(* IEC 61131-3 sources: SRCI/RobotLibrary/Library/POUs/BasicMove/MC_GroupInterrupt, 1 file *)

(* ---- MC_GroupInterruptFB.st ---- *)
/// Interrupt active movement, possible to continue movement
FUNCTION_BLOCK MC_GroupInterruptFB EXTENDS RobotLibraryBaseExecuteFB
// -------------------------------------------------------------------------
//  SRCI Robot Library
// -------------------------------------------------------------------------
//
//  Object:      GroupInterruptFB
//  Author:      Thorsten Brach
//  Date:        2024-06-01
//
//  Description:
//
//
//  Copyright:
//    (C) 2024 Thorsten Brach. All rights reserved
//             Licensed under the LGPL-3.0 license.
//
//  Disclaimer:
//    This project is provided without any guarantee and can be used for
//    private and commercial purposes. Any use is at the user’s
//    own risk and responsibility.
//
// -------------------------------------------------------------------------
VAR_INPUT
  /// Command parameter
  ParCmd          : GroupInterruptParCmd;
END_VAR

VAR_OUTPUT
  /// Command is transferred and confirmed by the RC
  CommandBuffered : BOOL;
  /// The command takes control of the motion of the according axis group.
  Active          : BOOL;
  /// Command output
  OutCmd          : GroupInterruptOutCmd;
END_VAR

VAR
  /// internal copy of command parameter
 _parCmd          : GroupInterruptParCmd;
  /// command data to send
 _command         : GroupInterruptSendData;
  /// response data received
 _response        : GroupInterruptRecvData;
END_VAR

  SUPER^(AxesGroup := AxesGroup);

END_FUNCTION_BLOCK

METHOD INTERNAL CheckAddParameter : BOOL
VAR_INPUT
  /// Payload pointer
  PayloadPtr : UDINT;
END_VAR
VAR
  /// Payload as byte array
  Payload    : ARRAY [1..SIZEOF(_command)] OF BYTE;
  /// Null Byte array
  Null       : ARRAY [1..SIZEOF(_command)] OF BYTE;
  /// Data length to compare
  DataLen    : UDINT;
END_VAR

  // Payload pointer must be decreased by one byte, because ADR(Payload) is already one byte !
  PayloadPtr := LIMIT (0, PayloadPtr - 1, SIZEOF(Payload) -1);
  // Convert command struct to payload array
  SysDepMemCpy( pDest := ADR(Payload), pSrc := ADR(_command), DataLen := SIZEOF(_command));
  // Calculate the data length to compare - at least one byte must be compared !
  DataLen := LIMIT(1, SIZEOF(Payload) - PayloadPtr, SIZEOF(Payload));
  // Compare Payload-Array with Null-Byte-Array
  CheckAddParameter := SysDepMemCmp( pData1 := ADR(Payload) + PayloadPtr , pData2 := ADR(Null), DataLen := DataLen) <>  RobotLibraryConstants.OK ;

END_METHOD

METHOD PROTECTED CheckFunctionSupported : BOOL
VAR_IN_OUT
  /// Robot assignment of function
  AxesGroup : AxesGroup;
END_VAR

  CheckFunctionSupported := AxesGroup.State.RobotData.RCSupportedFunctions.GroupInterrupt;

  IF ( NOT CheckFunctionSupported )
  THEN
    // call base implementation for set error and create log entry
    SUPER^.CheckFunctionSupported(AxesGroup := AxesGroup);
  END_IF

END_METHOD

METHOD PROTECTED CheckParameterChanged : BOOL
VAR_IN_OUT
  /// Robot assignment of function
  AxesGroup    : AxesGroup;
END_VAR

  // Check ParCmd Size is > 0, because MemCmp does not work correctly with size = 0
  IF (SIZEOF(ParCmd) = 0) OR (_stepCmd = 0)
  THEN
    RETURN;
  END_IF

  // compare memory
  _parameterChanged := ( SysDepMemCmp(pData1 := ADR(ParCmd), pData2 := ADR(_parCmd), DataLen := SIZEOF(ParCmd)) <> RobotLibraryConstants.OK );

  // check parameter valid ?
  _parameterValid   := CheckParameterValid( AxesGroup := AxesGroup );

  IF ((  _parameterChanged        )  AND
      (  _parameterValid          )) OR
      (  _parameterUpdateInternal )
  THEN
    // reset internal flag for send parameter update
   _parameterUpdateInternal := FALSE;
    // update internal copy of parameters
   _parCmd := ParCmd;
    // inc parameter sequence
   _command.ParSeq := _command.ParSeq + 1;
    // update command data
    CommandData := CreateCommandPayload(AxesGroup := AxesGroup); // ( Access via reference to rCommandFB in ACR )
    // notify active command register
    AxesGroup.Acyclic.ActiveCommandRegister.NotifyParameterChanged := _uniqueID;
  END_IF

END_METHOD

METHOD INTERNAL CreateCommandPayload : RobotLibraryCommandDataFB
VAR_IN_OUT
  /// Robot assignment of function
  AxesGroup : AxesGroup;
END_VAR
VAR
  /// Parameter count
 _parameterCnt : DINT;
END_VAR
// Table 6-273: Sent CMD payload (PLC to RC) of "GroupInterrupt"
// --------------------------
// Header
// --------------------------
// Byte 00 : UINT  - Type HB
// Byte 01 :       - Type LB
// Byte 02 : USINT - Reserve | ExecutionMode
// Byte 03 : USINT - ParSeq  | Priority
// --------------------------

  // set command parameter
  _command.CmdTyp     :=  CmdType.GroupInterrupt;
  _command.ExecMode   :=  ExecMode;
  _command.ParSeq     := _command.ParSeq;
  _command.Priority   :=  Priority;

  // copy command data to header
  _cmdHeader := _command;
  // call base implementation to copy header to payload buffer
  CreateCommandPayload := SUPER^.CreateCommandPayload(AxesGroup := AxesGroup);

  // Create logging
  CreateCommandPayloadLog(AxesGroup := AxesGroup, ParameterCnt := _parameterCnt);

END_METHOD

METHOD INTERNAL CreateCommandPayloadLog
VAR_IN_OUT
  /// Robot assignment of function
  AxesGroup : AxesGroup;
END_VAR
VAR_INPUT
  /// Parameter count
  ParameterCnt : DINT;
END_VAR

  // Create log entry for Parameter start
  CreateLogMessagePara1 ( Timestamp   := AxesGroup.State.SystemTime,
                          MessageType := MessageType.CMD,
                          Severity    := Severity.DEBUG,
                          MessageCode := 0,
                          MessageText := 'Create command payload with the {1} parameter(s) :',
                          Para1       := DINT_TO_STRING(ParameterCnt));

END_METHOD

METHOD FB_init : BOOL
VAR_INPUT
  /// if TRUE, the retain variables are initialized (warm start / cold start)
  bInitRetains : BOOL;
  /// if TRUE, the instance afterwards gets moved into the copy code (online change)
  bInCopyCode  : BOOL;
END_VAR

  MyType := 'MC_GroupInterruptFB';

  ExecMode := ExecutionMode.PARALLEL;
  Priority := PriorityLevel.NORMAL;

END_METHOD

METHOD PROTECTED OnExecRun : DINT
VAR_IN_OUT
  /// Robot assignment of function
  AxesGroup : AxesGroup;
END_VAR

  // call base implementation
  SUPER^.OnExecRun(AxesGroup := AxesGroup);

  CASE _stepCmd OF

    00:  IF ( _execute_R.Q ) AND ( NOT Error)
         THEN
           // Check function is supported and parameter are valid ?
           IF (( CheckFunctionSupported( AxesGroup := AxesGroup )) AND
               ( CheckParameterValid   ( AxesGroup := AxesGroup )))
           THEN
             // inc fast stop counter
             AxesGroup.Cyclic.PlcToRob.FastStop := AxesGroup.Cyclic.PlcToRob.FastStop + 1;
             // set busy flag
             Busy := TRUE;
             // Reset command outputs
             SysDepMemSet(pDest := ADR(OutCmd), Value := 0, DataLen := SIZEOF(OutCmd));
             // apply command parameter
            _parCmd := ParCmd;
             // init parameter sequence
            _command.ParSeq := 1;
             // create command data
             CommandData := CreateCommandPayload(AxesGroup := AxesGroup);
             // Add command to active command register
            _uniqueID := AxesGroup.Acyclic.ActiveCommandRegister.AddCmd( pCommandFB := ADR(THIS^ ));
             // set timeout
             SetTimeout(PT := _timeoutCmd, rTimer := _timerCmd);
             // inc step counter
            _stepCmd := _stepCmd + 1;
           END_IF
         END_IF

    01:  // Wait for responce received
         IF ( _responseReceived )
         THEN
           // reset response received flag
          _responseReceived := FALSE;
           // reset Active flag
           Active := FALSE;

           CASE  _response.State
           OF
             CmdMessageState.BUFFERED    : CommandBuffered := TRUE;
             CmdMessageState.ACTIVE      : Active          := TRUE;
             CmdMessageState.ERROR       : Error           := TRUE;
             CmdMessageState.DONE        : Done            := TRUE;

           END_CASE

           // Done, Aborted or Error ?
           IF (_response.State >= CmdMessageState.DONE )
           THEN
             // reset busy flag
             Busy := FALSE;
             // set timeout
             SetTimeout(PT := _timeoutCmd, rTimer := _timerCmd);
             // inc step counter
            _stepCmd := _stepCmd + 1;
           END_IF
         END_IF

    02: IF ( NOT Execute)
        THEN
          Reset();
        END_IF
  ELSE
    // invalid step
    ErrorID := RobotLibraryErrorIdEnum.ERR_INVALID_STEP;
  END_CASE

  // Reset FB
  IF ( NOT Execute )
  THEN
    Reset();
  END_IF

END_METHOD

METHOD INTERNAL ParseResponsePayload : DINT
VAR_INPUT
  /// Response data
  ResponseData : RobotLibraryResponseDataFB;
  /// Timestamp
  Timestamp    : SystemTime;
END_VAR
VAR
  /// Parameter count
 _parameterCnt : DINT;
END_VAR
// Table 6-274: Received CMD payload (RC to PLC) of "GroupInterrupt"
// --------------------------
// Header
// --------------------------
// Byte 00 : USINT - ParSeq | State
// Byte 01 : SINT  - AlarmMessageSeverity
// Byte 02 : UINT  - AlarmMessageCode HB
// Byte 03 :       - AlarmMessageCode LB

  // call base implementation to parse the header from payload buffer
  ResponseData.PayloadPtr := SUPER^.ParseResponsePayload(ResponseData := ResponseData, Timestamp := Timestamp);

  // copy parsed header to response
  _response.ParSeq               := _rspHeader.ParSeq;
  _response.State                := _rspHeader.State;
  _response.AlarmMessageSeverity := _rspHeader.AlarmMessageSeverity;
  _response.AlarmMessageCode     := _rspHeader.AlarmMessageCode;

  // Create logging
  ParseResponsePayloadLog(ResponseData := ResponseData, Timestamp := Timestamp, ParameterCnt := _parameterCnt);

END_METHOD

METHOD INTERNAL ParseResponsePayloadLog
VAR_INPUT
  /// Response data
  ResponseData : RobotLibraryResponseDataFB;
  /// Timestamp
  Timestamp    : SystemTime;
  /// Parameter count
  ParameterCnt : DINT;
END_VAR

  // Create log entry for Parameter start
  CreateLogMessagePara1 ( Timestamp   := Timestamp,
                          MessageType := MessageType.CMD,
                          Severity    := Severity.DEBUG,
                          MessageCode := 0,
                          MessageText := '{1} parameter(s) to parse from the response data:',
                          Para1       := DINT_TO_STRING(ParameterCnt));

  // Return if no parameter is remaining...
  IF ( ParameterCnt = 0 ) THEN RETURN; END_IF
  // dec remaining parameter(s)
  ParameterCnt := ParameterCnt - 1;
  // Create log entry for no parameter
  CreateLogMessage      ( Timestamp   := Timestamp,
                          MessageType := MessageType.CMD,
                          Severity    := Severity.DEBUG,
                          MessageCode := 0,
                          MessageText := 'This command has no parameter to parse...');

END_METHOD

METHOD PROTECTED Reset : DINT
VAR_INPUT
END_VAR

  Reset := SUPER^.Reset();

  Done               := FALSE;
  Busy               := FALSE;
  Active             := FALSE;
  CommandBuffered    := FALSE;

END_METHOD
